# EPICS substitutions: apps/db/user.substitutions
# Example substitutions file

file "db/dbExample1.db" {
    { user = "levon" }
}

file db/dbExample2.db {
    pattern { user, no, scan }
        { "levon", 1, "1 second" }
        { "levon", 2, "2 second" }
        { "levon", 3, "5 second" }
}
